ADAPTER ATurntable (* Adapter Interface *)
  (* Standard: 61499-1 *)
  (* Version 1.0, 2021-09-15, dorofeev *)
  (* Compiler header: package fb.test; *)
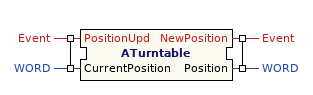
  EVENT_INPUT
    PositionUpd WITH CurrentPosition; (* Request from Socket *)
  END_EVENT
  EVENT_OUTPUT
    NewPosition WITH Position; (* Confirmation from Plug *)
  END_EVENT
  VAR_INPUT
    CurrentPosition : WORD; (* Request Data from Socket *)
  END_VAR
  VAR_OUTPUT
    Position : WORD; (* Confirmation Data from Plug *)
  END_VAR
  SERVICE PLUG/SOCKET (* Adapter Interface *)
    SEQUENCE request_confirm
      SOCKET.REQ(REQD) -> PLUG.REQ(REQD);
      PLUG.CNF(CNFD) -> SOCKET.CNF(CNFD);
    END_SEQUENCE
    SEQUENCE indication_response
      PLUG.IND(INDD) -> SOCKET.IND(INDD);
      SOCKET.RSP(RSPD) -> PLUG.RSP(RSPD);
    END_SEQUENCE
  END_SERVICE
END_ADAPTER
